FUNCTION_BLOCK VALUES2ARRAY_16_BYTE (* Service Interface Function Block Type *)
  (* Description: Copyright (c) 2014 Profactor GmbH This program and the accompanying materials are made available under the terms of the Eclipse Public License 2.0 which is available at https://www.eclipse.org/legal/epl-2.0/ SPDX-License-Identifier: EPL-2.0 *)
  (* Version 3.0, 2025-04-14, Patrick Aigner, changed package *)
  (* Version 1.0, 2014-07-09, Matthias Plasch, Profactor GmbH *)
  PACKAGE eclipse4diac::convert;
  {SET_ATTRIBUTE(eclipse4diac::core::GenericClassName, 'GEN_VALUES2ARRAY')}
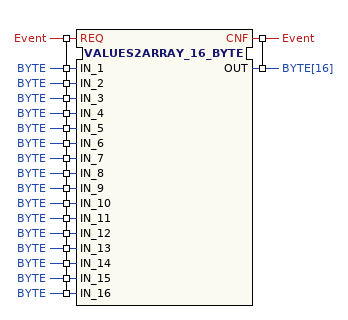
  EVENT_INPUT
    REQ WITH IN_1, IN_2, IN_3, IN_4, IN_5, IN_6, IN_7, IN_8, IN_9, IN_10, IN_11, IN_12, IN_13, IN_14, IN_15, IN_16; (* Service Request *)
  END_EVENT
  EVENT_OUTPUT
    CNF WITH OUT; (* Confirmation of Requested Service *)
  END_EVENT
  VAR_INPUT
    IN_1 : BYTE; (* input number 1 *)
    IN_2 : BYTE; (* input number 2 *)
    IN_3 : BYTE; (* input number 3 *)
    IN_4 : BYTE; (* input number 4 *)
    IN_5 : BYTE; (* input number 5 *)
    IN_6 : BYTE; (* input number 6 *)
    IN_7 : BYTE; (* input number 7 *)
    IN_8 : BYTE; (* input number 8 *)
    IN_9 : BYTE; (* input number 9 *)
    IN_10 : BYTE; (* input number 10 *)
    IN_11 : BYTE; (* input number 11 *)
    IN_12 : BYTE; (* input number 12 *)
    IN_13 : BYTE; (* input number 13 *)
    IN_14 : BYTE; (* input number 14 *)
    IN_15 : BYTE; (* input number 15 *)
    IN_16 : BYTE; (* input number 16 *)
  END_VAR
  VAR_OUTPUT
    OUT : ARRAY [0..15] OF BYTE; (* Array output *)
  END_VAR
END_FUNCTION_BLOCK
